FUNCTION_BLOCK ROBOTA1FB (* JADE WORKER *)
  (* Standard: 61499-1 *)
  (* Version 1.0, 2014-04-22, Ahmed, Fraunhofer IGD *)
  (* Compiler header: package fb.rt; *)
  (* Compiler Java Sun JDK 1.5.0 *)
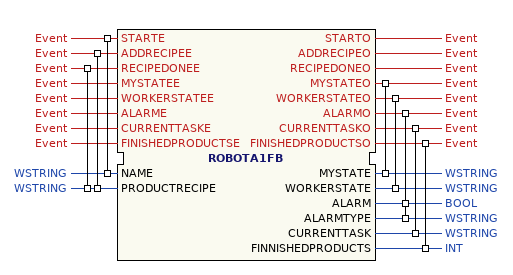
  EVENT_INPUT
    STARTE WITH NAME; (* Normal Execution Request *)
    ADDRECIPEE WITH PRODUCTRECIPE;
    RECIPEDONEE WITH PRODUCTRECIPE;
    MYSTATEE;
    WORKERSTATEE;
    ALARME;
    CURRENTTASKE;
    FINISHEDPRODUCTSE;
  END_EVENT
  EVENT_OUTPUT
    STARTO; (* Execution Confirmation *)
    ADDRECIPEO;
    RECIPEDONEO;
    MYSTATEO WITH MYSTATE;
    WORKERSTATEO WITH WORKERSTATE;
    ALARMO WITH ALARM, ALARMTYPE;
    CURRENTTASKO WITH CURRENTTASK;
    FINISHEDPRODUCTSO WITH FINNISHEDPRODUCTS;
  END_EVENT
  VAR_INPUT
    NAME : WSTRING;
    PRODUCTRECIPE : WSTRING;
  END_VAR
  VAR_OUTPUT
    MYSTATE : WSTRING;
    WORKERSTATE : WSTRING;
    ALARM : BOOL;
    ALARMTYPE : WSTRING;
    CURRENTTASK : WSTRING;
    FINNISHEDPRODUCTS : INT;
  END_VAR
END_FUNCTION_BLOCK
